// SIMATIC STEP 7 (V5.x) project Systemtest
// CPU: CPU 319-3 PN/DP
// station: Hardware
// station: SIMATIC 300
// station: P_ADR_BUS
// station: P_ADR_BUS
// station: Konfiguration
// station: SIMATIC PC Station
// program: S7-Programm(1)

SYMBOL_TABLE
"DB_FetchDATA"	DB 1	DB 1
"DB_WriteDATA"	DB 2	DB 2
"Connect_Param"	DB 211	DB 211
"FW_TCP"	FB 210	FB 210	// Fetch/Write via TCP
"FW_IOT"	FB 220	FB 220	// Fetch/Write via ISO on TCP
"RD_SINFO"	SFC 6	SFC 6	// Read OB Start Information
"BLKMOV"	SFC 20	SFC 20	// Copy Variables
"FILL"	SFC 21	SFC 21	// Initialize a Memory Area
"TEST_DB"	SFC 24	SFC 24	// Test Data Block
"STP"	SFC 46	SFC 46	// Change the CPU to STOP
"TSEND"	SFC 131	SFC 131	// Send Data
"TRCV"	SFC 132	SFC 132	// Receive Data
"TCON"	SFC 133	SFC 133	// Connect
"TDISCON"	SFC 134	SFC 134	// Disconnect
"T_USEND"	SFC 135	SFC 135
"T_URCV"	SFC 136	SFC 136
"VAT_FW"	VAT 1	
END_SYMBOL_TABLE
